(* CODESYS project MateusBastos_TalitaFelix_Versao_Final.project

Project tree, tasks and I/O mapping:
  Device : CODESYS Control Win V3, 3S - Smart Software Solutions GmbH, order no. 305021, version 3.5.11.40
    application Application
      libraries: Standard, * (System)
      task MainTask (cyclic, interval t#10ms, priority 1) calls Main_PGR
      global variables GVL
      Simulacao/
        Manual/
          program Manual_Simulacao_Silo_03 [ST]
          program Manual_Simulacao_Silo_02 [ST]
          program Manual_Simulacao_Silo_01 [ST]
        Automatico/
          program Doca2_Simulacao_Automatico [ST]
          program Doca1_Simulacao_Automatico [ST]
          program Valores_Doca2_Simulacao [ST]
          program Valores_Doca1_Simulacao [ST]
      Main/
        program Emergencia [ST]
        program Main_PGR [SFC]
      Docas/
        Manual/
          program Doca1_manual [SFC]
          program Doca2_manual [SFC]
        Automatico/
          program Doca1_automatico [SFC]
          program Doca2_automatico [SFC]
      program Alarmes [ST]
  program Valores_Simulacao_Manual [ST]
*)

// Device/Application/GVL
{attribute 'qualified_only'}
VAR_GLOBAL
// Sensores Analógicos - Entradas
LT_S01 : REAL;   // Sensor de porcentagem de etanol no silo 1
LT_S02 : REAL;   // Sensor de porcentagem de gasolina no silo 2
LT_S03 : REAL;   // Sensor de porcentagem de etanol no silo 3

// Sensores Discretos - Entradas
LSH_S01 : BOOL;  // Sensor de quantidade alta de combustível no silo 1
LSL_S01 : BOOL;  // Sensor de quantidade baixa de combustível no silo 1
LSH_S02 : BOOL;  // Sensor de quantidade alta de combustível no silo 2
LSL_S02 : BOOL;  // Sensor de quantidade baixa de combustível no silo 2
LSH_S03 : BOOL;  // Sensor de quantidade alta de combustível no silo 3
LSL_S03 : BOOL;  // Sensor de quantidade baixa de combustível no silo 3

ALARME_LSH_S01 : BOOL;  // Alarme de quantidade alta de combustível no silo 1
ALARME_LSL_S01 : BOOL;  // Alarme de quantidade baixa de combustível no silo 1
ALARME_LSH_S02 : BOOL;  // Alarme de quantidade alta de combustível no silo 2
ALARME_LSL_S02 : BOOL;  // Alarme de quantidade baixa de combustível no silo 2
ALARME_LSH_S03 : BOOL;  // Alarme de quantidade alta de combustível no silo 3
ALARME_LSL_S03 : BOOL;  // Alarme de quantidade baixa de combustível no silo 3

// Atuadores Discretos - Saídas
VA_S01 : BOOL;   // Válvula de admissão de etanol no silo 1
VA_S02 : BOOL;   // Válvula de admissão de gasolina no silo 2
VA_S03 : BOOL;   // Válvula de admissão de etanol no silo 3
VS_S01 : BOOL;   // Válvula de admissão de etanol no tanque
VS_S02_1 : BOOL; // Válvula de admissão de gasolina no tanque (primeira seção)
VS_S02_2 : BOOL; // Válvula de admissão de gasolina no tanque (segunda seção)
VS_S03 : BOOL;   // Válvula de admissão de etanol no tanque
VC_TQ2 : BOOL;   // Válvula de saída do combustível para a mangueira (tanque 2)
VC_TQ1 : BOOL;   // Válvula de saída do combustível para a mangueira (tanque 1)
M1 : BOOL;       // Misturador 1
M2 : BOOL;       // Misturador 2
B_R1 : BOOL;     // Bomba de Etanol
D1_B_R1 :BOOL;
D2_B_R1 :BOOL;
B_R2 : BOOL;
D1_B_R2 : BOOL;
D2_B_R2 : BOOL;     // Bomba de Gasolina
C_D1 : BOOL;     // Cancela 1
C_D2 : BOOL;     // Cancela 2

// Interface - máquina
liga: BOOL;
desliga: BOOL;
emergencia: BOOL;
rearme: BOOL;
Y_C_D1: BOOL;
Y_M_D1: BOOL;
Y_C_D2: BOOL;
Y_M_D2: BOOL;
etanol_D1: BOOL;
gasolina_p_D1: BOOL;
gasolina_n_D1: BOOL;
etanol_D2: BOOL;
gasolina_p_D2: BOOL;
gasolina_n_D2: BOOL;
//etanol_cheio: BOOL;
//gasolina_cheio: BOOL;
//timer_misturador: BOOL;
caminhao1_cheio: BOOL;
caminhao2_cheio: BOOL;
alarme_D1: BOOL;
alarme_D2: BOOL;

V_R_Etanol : INT := 100; //Vazao Reservatorio Etanol
V_R_Gasolina : INT := 100; //Vazao Reservatorio Gasolina
V_S01_TQ1 : INT := 50; // Vazão do Silo para o Tanque
V_S02_TQ : INT := 50; // Vazão DO Silo para o Tanque
V_S03_TQ2 : INT := 50; // Vazão DO Silo para o Tanque
TQ1_C : INT := 50;
TQ2_C : INT := 50;

volume_S01 : REAL := 50000;
volume_S02 : REAL := 50000;
volume_S03 : REAL := 50000;

volume_C1 : REAL := 0;
volume_C2 : REAL := 0;

volume_TQ1 : REAL := 0;
volume_TQ2 : REAL := 0;

volume_gasolina_C1 : REAL := 0;
volume_gasolina_C2 : REAL := 0;

volume_etanol_C1 : REAL := 0;
volume_etanol_C2 : REAL := 0;

PREMIUM : BOOL; 
ETANOL : BOOL; 

modo_op : BOOL; //Modo de operação atual do programa
switch : BOOl; //Modo de operação que o operador definiu

Transbordo_S03 : BOOL;
Transbordo_S02 : BOOL;
Transbordo_S01 : BOOL;

END_VAR

// Device/Application/Main/Main_PGR
PROGRAM Main_PGR
VAR
END_VAR

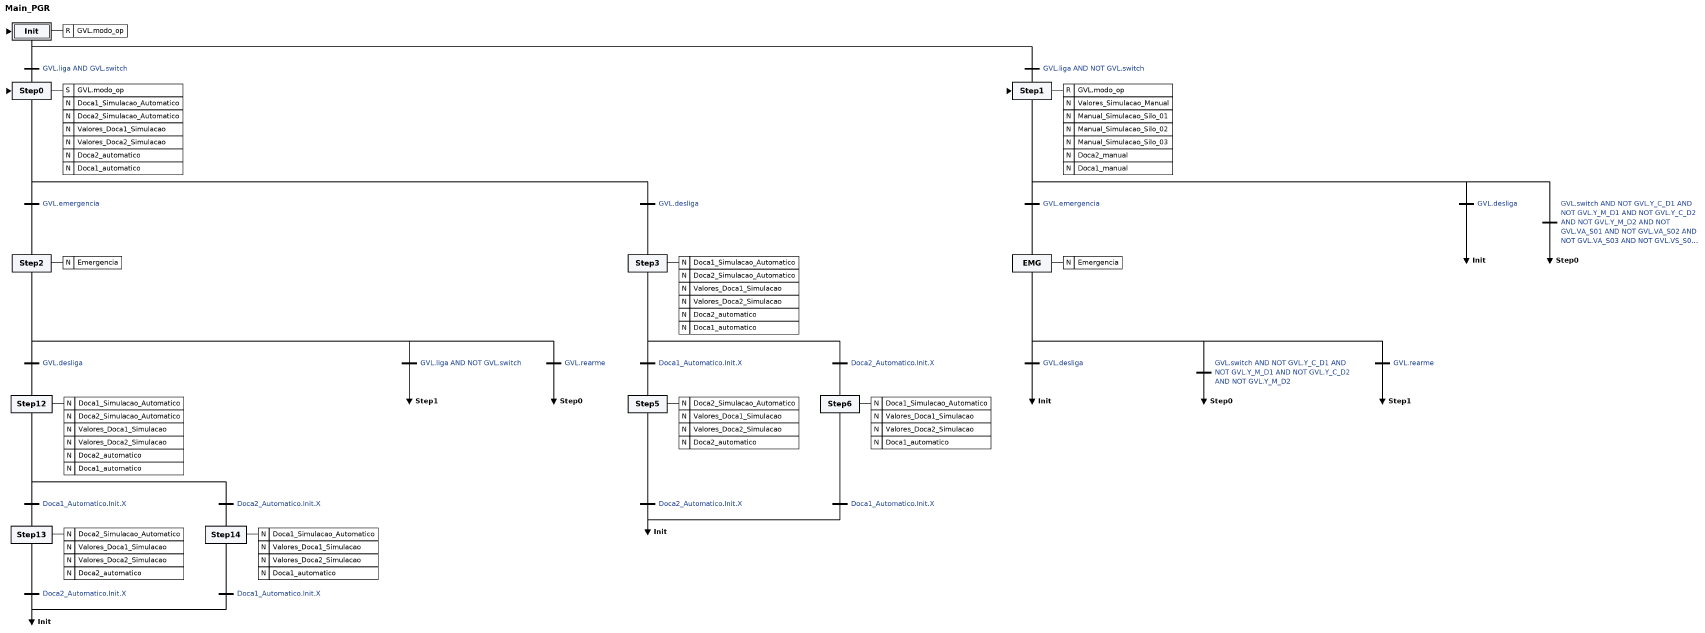
INITIAL_STEP Init:
    GVL.modo_op(R);
END_STEP
TRANSITION FROM Init TO Step0
    := GVL.liga AND GVL.switch;
END_TRANSITION
STEP Step0:
    GVL.modo_op(S);
    Doca1_Simulacao_Automatico(N);
    Doca2_Simulacao_Automatico(N);
    Valores_Doca1_Simulacao(N);
    Valores_Doca2_Simulacao(N);
    Doca2_automatico(N);
    Doca1_automatico(N);
END_STEP
TRANSITION FROM Step0 TO Step2
    := GVL.emergencia;
END_TRANSITION
STEP Step2:
    Emergencia(N);
END_STEP
TRANSITION FROM Step2 TO Step12
    := GVL.desliga;
END_TRANSITION
TRANSITION FROM Step2 TO Step1
    := GVL.liga AND NOT GVL.switch;
END_TRANSITION
TRANSITION FROM Step2 TO Step0
    := GVL.rearme;
END_TRANSITION
TRANSITION FROM Step0 TO Step3
    := GVL.desliga;
END_TRANSITION
STEP Step3:
    Doca1_Simulacao_Automatico(N);
    Doca2_Simulacao_Automatico(N);
    Valores_Doca1_Simulacao(N);
    Valores_Doca2_Simulacao(N);
    Doca2_automatico(N);
    Doca1_automatico(N);
END_STEP
TRANSITION FROM Step3 TO Step5
    := Doca1_Automatico.Init.X;
END_TRANSITION
STEP Step5:
    Doca2_Simulacao_Automatico(N);
    Valores_Doca1_Simulacao(N);
    Valores_Doca2_Simulacao(N);
    Doca2_automatico(N);
END_STEP
TRANSITION FROM Step5 TO Init
    := Doca2_Automatico.Init.X;
END_TRANSITION
TRANSITION FROM Step3 TO Step6
    := Doca2_Automatico.Init.X;
END_TRANSITION
STEP Step6:
    Doca1_Simulacao_Automatico(N);
    Valores_Doca1_Simulacao(N);
    Valores_Doca2_Simulacao(N);
    Doca1_automatico(N);
END_STEP
TRANSITION FROM Step6 TO Init
    := Doca1_Automatico.Init.X;
END_TRANSITION
TRANSITION FROM Init TO Step1
    := GVL.liga AND NOT GVL.switch;
END_TRANSITION
STEP Step1:
    GVL.modo_op(R);
    Valores_Simulacao_Manual(N);
    Manual_Simulacao_Silo_01(N);
    Manual_Simulacao_Silo_02(N);
    Manual_Simulacao_Silo_03(N);
    Doca2_manual(N);
    Doca1_manual(N);
END_STEP
TRANSITION FROM Step1 TO EMG
    := GVL.emergencia;
END_TRANSITION
STEP EMG:
    Emergencia(N);
END_STEP
TRANSITION FROM Step1 TO Init
    := GVL.desliga;
END_TRANSITION
TRANSITION FROM Step1 TO Step0
    := GVL.switch AND NOT GVL.Y_C_D1 AND NOT GVL.Y_M_D1 AND NOT GVL.Y_C_D2 AND NOT GVL.Y_M_D2 AND NOT GVL.VA_S01 AND NOT GVL.VA_S02 AND NOT GVL.VA_S03 AND NOT GVL.VS_S01 AND NOT GVL.VS_S02_1 AND NOT GVL.VS_S02_2 AND NOT GVL.VS_S03 AND NOT GVL.VC_TQ2 AND NOT GVL.VC_TQ1 AND NOT GVL.B_R2 AND NOT GVL.B_R1 AND NOT GVL.M1 AND NOT GVL.M2;
END_TRANSITION
TRANSITION FROM EMG TO Init
    := GVL.desliga;
END_TRANSITION
TRANSITION FROM EMG TO Step0
    := GVL.switch AND NOT GVL.Y_C_D1 AND NOT GVL.Y_M_D1 AND NOT GVL.Y_C_D2 AND NOT GVL.Y_M_D2;
END_TRANSITION
TRANSITION FROM EMG TO Step1
    := GVL.rearme;
END_TRANSITION
STEP Step12:
    Doca1_Simulacao_Automatico(N);
    Doca2_Simulacao_Automatico(N);
    Valores_Doca1_Simulacao(N);
    Valores_Doca2_Simulacao(N);
    Doca2_automatico(N);
    Doca1_automatico(N);
END_STEP
TRANSITION FROM Step12 TO Step13
    := Doca1_Automatico.Init.X;
END_TRANSITION
STEP Step13:
    Doca2_Simulacao_Automatico(N);
    Valores_Doca1_Simulacao(N);
    Valores_Doca2_Simulacao(N);
    Doca2_automatico(N);
END_STEP
TRANSITION FROM Step13 TO Init
    := Doca2_Automatico.Init.X;
END_TRANSITION
TRANSITION FROM Step12 TO Step14
    := Doca2_Automatico.Init.X;
END_TRANSITION
STEP Step14:
    Doca1_Simulacao_Automatico(N);
    Valores_Doca1_Simulacao(N);
    Valores_Doca2_Simulacao(N);
    Doca1_automatico(N);
END_STEP
TRANSITION FROM Step14 TO Init
    := Doca1_Automatico.Init.X;
END_TRANSITION

END_PROGRAM

// Device/Application/Simulacao/Automatico/Doca2_Simulacao_Automatico
PROGRAM Doca2_Simulacao_Automatico
VAR
END_VAR

IF NOT GVL.emergencia AND GVL.switch THEN
	//Estado  20 & //Estado 31 & //Estado 41 & //Estado 34 & //Estado 44
	IF GVL.VA_S03 AND GVL.D2_B_R1 AND NOT GVL.LSH_S03 THEN
	// Enchendo o Silo 01 de Etanol - STEP_21
		GVL.volume_S03 := GVL.volume_S03 + GVL.V_R_Etanol;
	
		GVL.volume_TQ2 := GVL.volume_TQ2;
		
		GVL.volume_C2 := GVL.volume_C2;
		
	//Estado  20	
	ELSIF GVL.VA_S02 AND (GVL.D1_B_R2 OR GVL.D2_B_R2) AND (GVL.ETANOL OR NOT GVL.Y_C_D1) AND NOT GVL.LSH_S02 THEN // Caso em que o somente a doca 2 está utilizando gasolina
		GVL.volume_S02 := GVL.volume_S02 + GVL.V_R_Gasolina;
		
	ELSIF GVL.VS_S03 AND GVL.C_D2 AND NOT GVL.VS_S02_2 AND GVL.VC_TQ2 AND GVL.volume_S03 > 0 THEN
	// Enchendo o Tanque 1 & Esvaziando o Silo 01 - STEP_20
		GVL.volume_S03 := GVL.volume_S03 - GVL.V_S03_TQ2;
		
		GVL.volume_TQ2 := GVL.volume_TQ2 + GVL.TQ2_C - GVL.V_S03_TQ2;
		
		GVL.volume_C2 := GVL.volume_C2 + GVL.TQ2_C;
		
	//Estado 30	- STEP_30 e STEP_40
	ELSIF GVL.VS_S03 AND GVL.VS_S02_2 AND GVL.C_D2 AND GVL.volume_S03 > 0 AND GVL.volume_S02 > 0 THEN
	// Enchendo o TQ 1 && Esvaziando o Silo 01 && Esvaziando o Silo 02
	
	//Situação em que começo a encher o tanque de gasolina e de etanol simultaneamente
	
		GVL.volume_S03 := GVL.volume_S03 - GVL.V_S03_TQ2; // Diminuo o volume do Silo 3
		
		GVL.volume_S02 := GVL.volume_S02 - GVL.V_S02_TQ; // Diminuo o volume do Silo 2
		
		GVL.volume_C2 := GVL.volume_C2; // Mantenho o volume do caminhão constante
		
		GVL.volume_TQ2 := GVL.volume_TQ2 + GVL.V_S02_TQ + GVL.V_S03_TQ2; // Aumento o volume do tanque 1
		
		GVL.volume_gasolina_C2 := GVL.volume_gasolina_C2 + GVL.V_S02_TQ; // Aumento a contagem da gasolina que está entrando no tanque
		
		GVL.volume_etanol_C2 := GVL.volume_etanol_C2 + GVL.V_S03_TQ2; // Aumento a contagem de etanol que está entrando no tanque
		
	//Estado 33 & Estado 43 - STEP_33
	ELSIF GVL.VS_S02_2 AND NOT GVL.VC_TQ2 AND GVL.C_D2 AND GVL.volume_S02 > 0 THEN
		GVL.volume_S02 := GVL.volume_S02 - GVL.V_S02_TQ;	
		
		GVL.volume_C2 := GVL.volume_C2;
		
		GVL.volume_TQ2 := GVL.volume_TQ2 + GVL.V_S02_TQ;
		
		GVL.volume_gasolina_C2 := GVL.volume_gasolina_C2 + GVL.V_S02_TQ;
		
	//Estado 35 & //Estado 45
	ELSIF GVL.M2 AND GVL.C_D2 THEN
		GVL.volume_C2 := GVL.volume_C2;
		GVL.volume_TQ2 := GVL.volume_TQ2;
		
	//Estado 36 & //Estado 46
	ELSIF GVL.VC_TQ2 AND GVL.C_D2 AND GVL.volume_TQ2 > 0 THEN
		GVL.volume_C2 := GVL.volume_C2 + GVL.TQ2_C;
		GVL.volume_TQ2 := GVL.volume_TQ2 - GVL.TQ2_C;
	
	ELSIF NOT GVL.Y_C_D2 AND NOT GVL.C_D2 THEN 
		GVL.volume_C2 := 0;
		GVL.volume_TQ2 := 0;
		
		Doca2_automatico.gasolina_cheio := FALSE;
		Doca2_automatico.etanol_cheio := FALSE;
		GVL.caminhao2_cheio := FALSE;
	
	END_IF
END_IF

END_PROGRAM

// Device/Application/Main/Emergencia
PROGRAM Emergencia


	GVL.VA_S01 := FALSE;   
	GVL.VA_S02 := FALSE;
	GVL.VA_S03 := FALSE;
	GVL.VS_S01 := FALSE;
	GVL.VS_S02_1 := FALSE;
	GVL.VS_S02_2 := FALSE;
	GVL.VS_S03 := FALSE;
	GVL.VC_TQ2 := FALSE;
	GVL.VC_TQ1 := FALSE;
	GVL.M1 := FALSE;
	GVL.M2 := FALSE;

END_PROGRAM

// Device/Application/Docas/Automatico/Doca2_automatico
PROGRAM Doca2_automatico
VAR_INPUT
	etanol_cheio: BOOL;
	gasolina_cheio: BOOL;
END_VAR

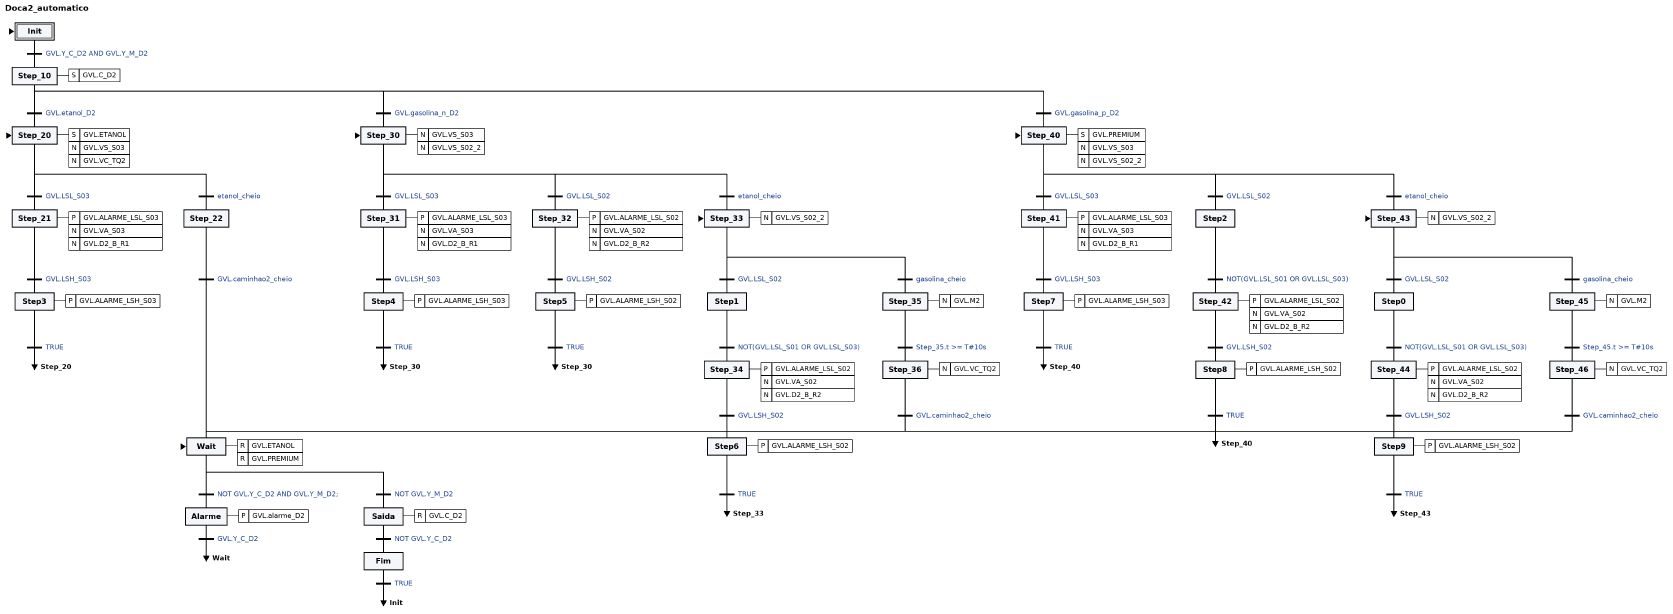
INITIAL_STEP Init:
END_STEP
TRANSITION FROM Init TO Step_10
    := GVL.Y_C_D2 AND GVL.Y_M_D2;
END_TRANSITION
STEP Step_10:
    GVL.C_D2(S);
END_STEP
TRANSITION FROM Step_10 TO Step_20
    := GVL.etanol_D2;
END_TRANSITION
STEP Step_20:
    GVL.ETANOL(S);
    GVL.VS_S03(N);
    GVL.VC_TQ2(N);
END_STEP
TRANSITION FROM Step_20 TO Step_21
    := GVL.LSL_S03;
END_TRANSITION
STEP Step_21:
    GVL.ALARME_LSL_S03(P);
    GVL.VA_S03(N);
    GVL.D2_B_R1(N);
END_STEP
TRANSITION FROM Step_21 TO Step3
    := GVL.LSH_S03;
END_TRANSITION
STEP Step3:
    GVL.ALARME_LSH_S03(P);
END_STEP
TRANSITION FROM Step3 TO Step_20
    := TRUE;
END_TRANSITION
TRANSITION FROM Step_20 TO Step_22
    := etanol_cheio;
END_TRANSITION
STEP Step_22:
END_STEP
TRANSITION FROM Step_22 TO Wait
    := GVL.caminhao2_cheio;
END_TRANSITION
TRANSITION FROM Step_10 TO Step_30
    := GVL.gasolina_n_D2;
END_TRANSITION
STEP Step_30:
    GVL.VS_S03(N);
    GVL.VS_S02_2(N);
END_STEP
TRANSITION FROM Step_30 TO Step_31
    := GVL.LSL_S03;
END_TRANSITION
STEP Step_31:
    GVL.ALARME_LSL_S03(P);
    GVL.VA_S03(N);
    GVL.D2_B_R1(N);
END_STEP
TRANSITION FROM Step_31 TO Step4
    := GVL.LSH_S03;
END_TRANSITION
STEP Step4:
    GVL.ALARME_LSH_S03(P);
END_STEP
TRANSITION FROM Step4 TO Step_30
    := TRUE;
END_TRANSITION
TRANSITION FROM Step_30 TO Step_32
    := GVL.LSL_S02;
END_TRANSITION
STEP Step_32:
    GVL.ALARME_LSL_S02(P);
    GVL.VA_S02(N);
    GVL.D2_B_R2(N);
END_STEP
TRANSITION FROM Step_32 TO Step5
    := GVL.LSH_S02;
END_TRANSITION
STEP Step5:
    GVL.ALARME_LSH_S02(P);
END_STEP
TRANSITION FROM Step5 TO Step_30
    := TRUE;
END_TRANSITION
TRANSITION FROM Step_30 TO Step_33
    := etanol_cheio;
END_TRANSITION
STEP Step_33:
    GVL.VS_S02_2(N);
END_STEP
TRANSITION FROM Step_33 TO Step1
    := GVL.LSL_S02;
END_TRANSITION
STEP Step1:
END_STEP
TRANSITION FROM Step1 TO Step_34
    := NOT(GVL.LSL_S01 OR GVL.LSL_S03);
END_TRANSITION
STEP Step_34:
    GVL.ALARME_LSL_S02(P);
    GVL.VA_S02(N);
    GVL.D2_B_R2(N);
END_STEP
TRANSITION FROM Step_34 TO Step6
    := GVL.LSH_S02;
END_TRANSITION
STEP Step6:
    GVL.ALARME_LSH_S02(P);
END_STEP
TRANSITION FROM Step6 TO Step_33
    := TRUE;
END_TRANSITION
TRANSITION FROM Step_33 TO Step_35
    := gasolina_cheio;
END_TRANSITION
STEP Step_35:
    GVL.M2(N);
END_STEP
TRANSITION FROM Step_35 TO Step_36
    := Step_35.t >= T#10s;
END_TRANSITION
STEP Step_36:
    GVL.VC_TQ2(N);
END_STEP
TRANSITION FROM Step_36 TO Wait
    := GVL.caminhao2_cheio;
END_TRANSITION
TRANSITION FROM Step_10 TO Step_40
    := GVL.gasolina_p_D2;
END_TRANSITION
STEP Step_40:
    GVL.PREMIUM(S);
    GVL.VS_S03(N);
    GVL.VS_S02_2(N);
END_STEP
TRANSITION FROM Step_40 TO Step_41
    := GVL.LSL_S03;
END_TRANSITION
STEP Step_41:
    GVL.ALARME_LSL_S03(P);
    GVL.VA_S03(N);
    GVL.D2_B_R1(N);
END_STEP
TRANSITION FROM Step_41 TO Step7
    := GVL.LSH_S03;
END_TRANSITION
STEP Step7:
    GVL.ALARME_LSH_S03(P);
END_STEP
TRANSITION FROM Step7 TO Step_40
    := TRUE;
END_TRANSITION
TRANSITION FROM Step_40 TO Step2
    := GVL.LSL_S02;
END_TRANSITION
STEP Step2:
END_STEP
TRANSITION FROM Step2 TO Step_42
    := NOT(GVL.LSL_S01 OR GVL.LSL_S03);
END_TRANSITION
STEP Step_42:
    GVL.ALARME_LSL_S02(P);
    GVL.VA_S02(N);
    GVL.D2_B_R2(N);
END_STEP
TRANSITION FROM Step_42 TO Step8
    := GVL.LSH_S02;
END_TRANSITION
STEP Step8:
    GVL.ALARME_LSH_S02(P);
END_STEP
TRANSITION FROM Step8 TO Step_40
    := TRUE;
END_TRANSITION
TRANSITION FROM Step_40 TO Step_43
    := etanol_cheio;
END_TRANSITION
STEP Step_43:
    GVL.VS_S02_2(N);
END_STEP
TRANSITION FROM Step_43 TO Step0
    := GVL.LSL_S02;
END_TRANSITION
STEP Step0:
END_STEP
TRANSITION FROM Step0 TO Step_44
    := NOT(GVL.LSL_S01 OR GVL.LSL_S03);
END_TRANSITION
STEP Step_44:
    GVL.ALARME_LSL_S02(P);
    GVL.VA_S02(N);
    GVL.D2_B_R2(N);
END_STEP
TRANSITION FROM Step_44 TO Step9
    := GVL.LSH_S02;
END_TRANSITION
STEP Step9:
    GVL.ALARME_LSH_S02(P);
END_STEP
TRANSITION FROM Step9 TO Step_43
    := TRUE;
END_TRANSITION
TRANSITION FROM Step_43 TO Step_45
    := gasolina_cheio;
END_TRANSITION
STEP Step_45:
    GVL.M2(N);
END_STEP
TRANSITION FROM Step_45 TO Step_46
    := Step_45.t >= T#10s;
END_TRANSITION
STEP Step_46:
    GVL.VC_TQ2(N);
END_STEP
TRANSITION FROM Step_46 TO Wait
    := GVL.caminhao2_cheio;
END_TRANSITION
STEP Wait:
    GVL.ETANOL(R);
    GVL.PREMIUM(R);
END_STEP
TRANSITION FROM Wait TO Alarme
    := NOT GVL.Y_C_D2 AND GVL.Y_M_D2;
END_TRANSITION
STEP Alarme:
    GVL.alarme_D2(P);
END_STEP
TRANSITION FROM Alarme TO Wait
    := GVL.Y_C_D2;
END_TRANSITION
TRANSITION FROM Wait TO Saida
    := NOT GVL.Y_M_D2;
END_TRANSITION
STEP Saida:
    GVL.C_D2(R);
END_STEP
TRANSITION FROM Saida TO Fim
    := NOT GVL.Y_C_D2;
END_TRANSITION
STEP Fim:
END_STEP
TRANSITION FROM Fim TO Init
    := TRUE;
END_TRANSITION

END_PROGRAM

// Device/Application/Docas/Manual/Doca1_manual
PROGRAM Doca1_manual
VAR_INPUT
	Ligar : BOOL;
END_VAR

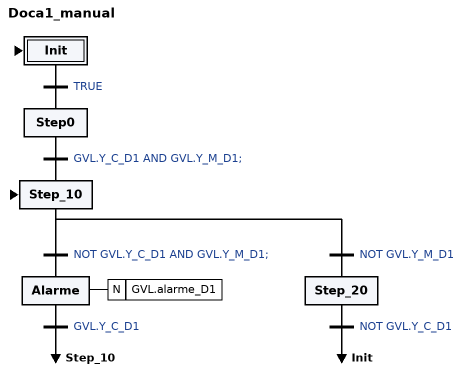
INITIAL_STEP Init:
END_STEP
TRANSITION FROM Init TO Step0
    := TRUE;
END_TRANSITION
STEP Step0:
END_STEP
TRANSITION FROM Step0 TO Step_10
    := GVL.Y_C_D1 AND GVL.Y_M_D1;
END_TRANSITION
STEP Step_10:
END_STEP
TRANSITION FROM Step_10 TO Alarme
    := NOT GVL.Y_C_D1 AND GVL.Y_M_D1;
END_TRANSITION
STEP Alarme:
    GVL.alarme_D1(N);
END_STEP
TRANSITION FROM Alarme TO Step_10
    := GVL.Y_C_D1;
END_TRANSITION
TRANSITION FROM Step_10 TO Step_20
    := NOT GVL.Y_M_D1;
END_TRANSITION
STEP Step_20:
END_STEP
TRANSITION FROM Step_20 TO Init
    := NOT GVL.Y_C_D1;
END_TRANSITION

END_PROGRAM

// Device/Application/Docas/Manual/Doca2_manual
PROGRAM Doca2_manual

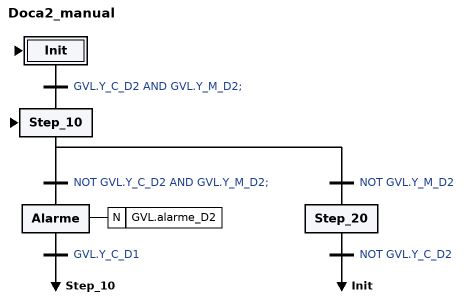
INITIAL_STEP Init:
END_STEP
TRANSITION FROM Init TO Step_10
    := GVL.Y_C_D2 AND GVL.Y_M_D2;
END_TRANSITION
STEP Step_10:
END_STEP
TRANSITION FROM Step_10 TO Alarme
    := NOT GVL.Y_C_D2 AND GVL.Y_M_D2;
END_TRANSITION
STEP Alarme:
    GVL.alarme_D2(N);
END_STEP
TRANSITION FROM Alarme TO Step_10
    := GVL.Y_C_D1;
END_TRANSITION
TRANSITION FROM Step_10 TO Step_20
    := NOT GVL.Y_M_D2;
END_TRANSITION
STEP Step_20:
END_STEP
TRANSITION FROM Step_20 TO Init
    := NOT GVL.Y_C_D2;
END_TRANSITION

END_PROGRAM

// Device/Application/Docas/Automatico/Doca1_automatico
PROGRAM Doca1_automatico

VAR_INPUT
	etanol_cheio: BOOL;
	gasolina_cheio: BOOL;
END_VAR

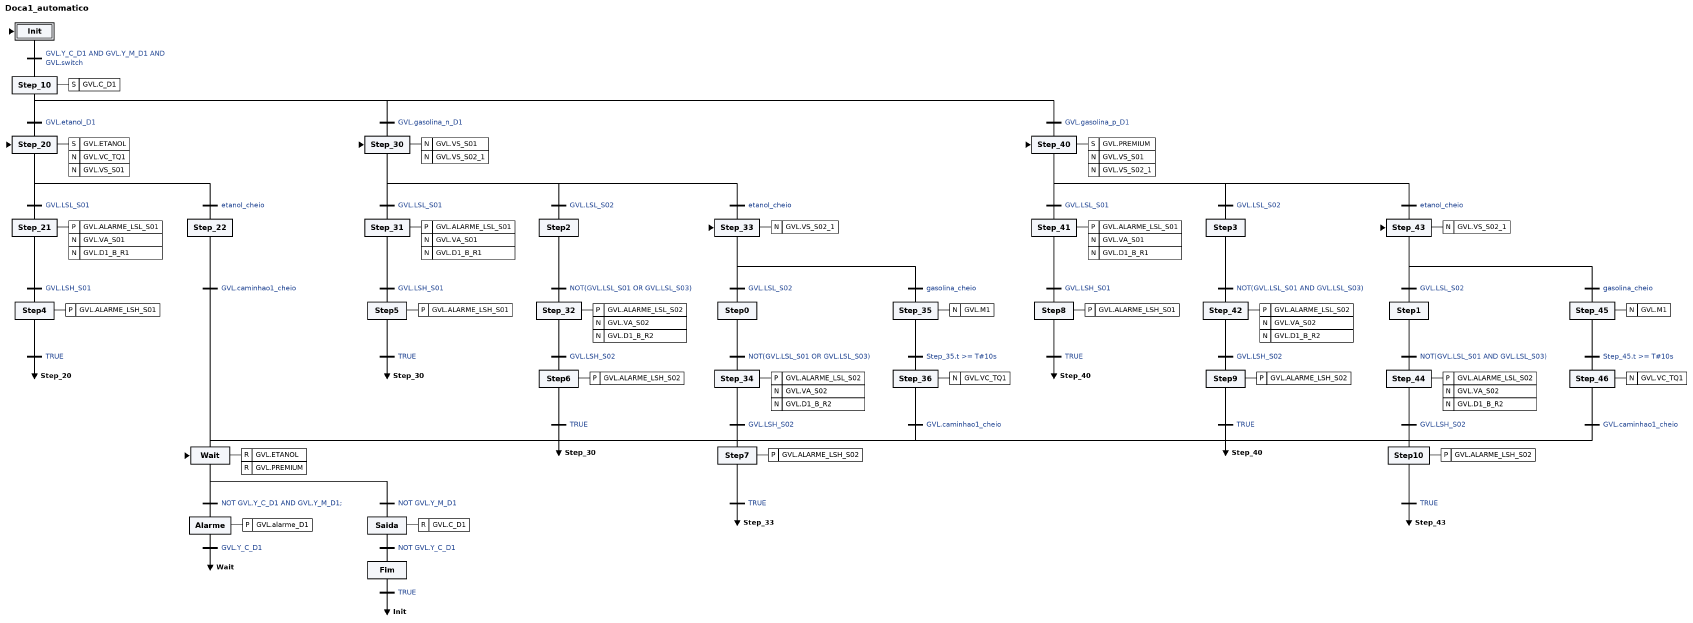
INITIAL_STEP Init:
END_STEP
TRANSITION FROM Init TO Step_10
    := GVL.Y_C_D1 AND GVL.Y_M_D1 AND GVL.switch;
END_TRANSITION
STEP Step_10:
    GVL.C_D1(S);
END_STEP
TRANSITION FROM Step_10 TO Step_20
    := GVL.etanol_D1;
END_TRANSITION
STEP Step_20:
    GVL.ETANOL(S);
    GVL.VC_TQ1(N);
    GVL.VS_S01(N);
END_STEP
TRANSITION FROM Step_20 TO Step_21
    := GVL.LSL_S01;
END_TRANSITION
STEP Step_21:
    GVL.ALARME_LSL_S01(P);
    GVL.VA_S01(N);
    GVL.D1_B_R1(N);
END_STEP
TRANSITION FROM Step_21 TO Step4
    := GVL.LSH_S01;
END_TRANSITION
STEP Step4:
    GVL.ALARME_LSH_S01(P);
END_STEP
TRANSITION FROM Step4 TO Step_20
    := TRUE;
END_TRANSITION
TRANSITION FROM Step_20 TO Step_22
    := etanol_cheio;
END_TRANSITION
STEP Step_22:
END_STEP
TRANSITION FROM Step_22 TO Wait
    := GVL.caminhao1_cheio;
END_TRANSITION
TRANSITION FROM Step_10 TO Step_30
    := GVL.gasolina_n_D1;
END_TRANSITION
STEP Step_30:
    GVL.VS_S01(N);
    GVL.VS_S02_1(N);
END_STEP
TRANSITION FROM Step_30 TO Step_31
    := GVL.LSL_S01;
END_TRANSITION
STEP Step_31:
    GVL.ALARME_LSL_S01(P);
    GVL.VA_S01(N);
    GVL.D1_B_R1(N);
END_STEP
TRANSITION FROM Step_31 TO Step5
    := GVL.LSH_S01;
END_TRANSITION
STEP Step5:
    GVL.ALARME_LSH_S01(P);
END_STEP
TRANSITION FROM Step5 TO Step_30
    := TRUE;
END_TRANSITION
TRANSITION FROM Step_30 TO Step2
    := GVL.LSL_S02;
END_TRANSITION
STEP Step2:
END_STEP
TRANSITION FROM Step2 TO Step_32
    := NOT(GVL.LSL_S01 OR GVL.LSL_S03);
END_TRANSITION
STEP Step_32:
    GVL.ALARME_LSL_S02(P);
    GVL.VA_S02(N);
    GVL.D1_B_R2(N);
END_STEP
TRANSITION FROM Step_32 TO Step6
    := GVL.LSH_S02;
END_TRANSITION
STEP Step6:
    GVL.ALARME_LSH_S02(P);
END_STEP
TRANSITION FROM Step6 TO Step_30
    := TRUE;
END_TRANSITION
TRANSITION FROM Step_30 TO Step_33
    := etanol_cheio;
END_TRANSITION
STEP Step_33:
    GVL.VS_S02_1(N);
END_STEP
TRANSITION FROM Step_33 TO Step0
    := GVL.LSL_S02;
END_TRANSITION
STEP Step0:
END_STEP
TRANSITION FROM Step0 TO Step_34
    := NOT(GVL.LSL_S01 OR GVL.LSL_S03);
END_TRANSITION
STEP Step_34:
    GVL.ALARME_LSL_S02(P);
    GVL.VA_S02(N);
    GVL.D1_B_R2(N);
END_STEP
TRANSITION FROM Step_34 TO Step7
    := GVL.LSH_S02;
END_TRANSITION
STEP Step7:
    GVL.ALARME_LSH_S02(P);
END_STEP
TRANSITION FROM Step7 TO Step_33
    := TRUE;
END_TRANSITION
TRANSITION FROM Step_33 TO Step_35
    := gasolina_cheio;
END_TRANSITION
STEP Step_35:
    GVL.M1(N);
END_STEP
TRANSITION FROM Step_35 TO Step_36
    := Step_35.t >= T#10s;
END_TRANSITION
STEP Step_36:
    GVL.VC_TQ1(N);
END_STEP
TRANSITION FROM Step_36 TO Wait
    := GVL.caminhao1_cheio;
END_TRANSITION
TRANSITION FROM Step_10 TO Step_40
    := GVL.gasolina_p_D1;
END_TRANSITION
STEP Step_40:
    GVL.PREMIUM(S);
    GVL.VS_S01(N);
    GVL.VS_S02_1(N);
END_STEP
TRANSITION FROM Step_40 TO Step_41
    := GVL.LSL_S01;
END_TRANSITION
STEP Step_41:
    GVL.ALARME_LSL_S01(P);
    GVL.VA_S01(N);
    GVL.D1_B_R1(N);
END_STEP
TRANSITION FROM Step_41 TO Step8
    := GVL.LSH_S01;
END_TRANSITION
STEP Step8:
    GVL.ALARME_LSH_S01(P);
END_STEP
TRANSITION FROM Step8 TO Step_40
    := TRUE;
END_TRANSITION
TRANSITION FROM Step_40 TO Step3
    := GVL.LSL_S02;
END_TRANSITION
STEP Step3:
END_STEP
TRANSITION FROM Step3 TO Step_42
    := NOT(GVL.LSL_S01 AND GVL.LSL_S03);
END_TRANSITION
STEP Step_42:
    GVL.ALARME_LSL_S02(P);
    GVL.VA_S02(N);
    GVL.D1_B_R2(N);
END_STEP
TRANSITION FROM Step_42 TO Step9
    := GVL.LSH_S02;
END_TRANSITION
STEP Step9:
    GVL.ALARME_LSH_S02(P);
END_STEP
TRANSITION FROM Step9 TO Step_40
    := TRUE;
END_TRANSITION
TRANSITION FROM Step_40 TO Step_43
    := etanol_cheio;
END_TRANSITION
STEP Step_43:
    GVL.VS_S02_1(N);
END_STEP
TRANSITION FROM Step_43 TO Step1
    := GVL.LSL_S02;
END_TRANSITION
STEP Step1:
END_STEP
TRANSITION FROM Step1 TO Step_44
    := NOT(GVL.LSL_S01 AND GVL.LSL_S03);
END_TRANSITION
STEP Step_44:
    GVL.ALARME_LSL_S02(P);
    GVL.VA_S02(N);
    GVL.D1_B_R2(N);
END_STEP
TRANSITION FROM Step_44 TO Step10
    := GVL.LSH_S02;
END_TRANSITION
STEP Step10:
    GVL.ALARME_LSH_S02(P);
END_STEP
TRANSITION FROM Step10 TO Step_43
    := TRUE;
END_TRANSITION
TRANSITION FROM Step_43 TO Step_45
    := gasolina_cheio;
END_TRANSITION
STEP Step_45:
    GVL.M1(N);
END_STEP
TRANSITION FROM Step_45 TO Step_46
    := Step_45.t >= T#10s;
END_TRANSITION
STEP Step_46:
    GVL.VC_TQ1(N);
END_STEP
TRANSITION FROM Step_46 TO Wait
    := GVL.caminhao1_cheio;
END_TRANSITION
STEP Wait:
    GVL.ETANOL(R);
    GVL.PREMIUM(R);
END_STEP
TRANSITION FROM Wait TO Alarme
    := NOT GVL.Y_C_D1 AND GVL.Y_M_D1;
END_TRANSITION
STEP Alarme:
    GVL.alarme_D1(P);
END_STEP
TRANSITION FROM Alarme TO Wait
    := GVL.Y_C_D1;
END_TRANSITION
TRANSITION FROM Wait TO Saida
    := NOT GVL.Y_M_D1;
END_TRANSITION
STEP Saida:
    GVL.C_D1(R);
END_STEP
TRANSITION FROM Saida TO Fim
    := NOT GVL.Y_C_D1;
END_TRANSITION
STEP Fim:
END_STEP
TRANSITION FROM Fim TO Init
    := TRUE;
END_TRANSITION

END_PROGRAM

// Device/Application/Simulacao/Manual/Manual_Simulacao_Silo_03
PROGRAM Manual_Simulacao_Silo_03
VAR
END_VAR

IF NOT GVL.emergencia AND NOT GVL.switch THEN
	
	IF NOT GVL.D1_B_R1 AND NOT GVL.VS_S03 AND GVL.VC_TQ2 THEN
	
		IF GVL.volume_TQ2 > 0 THEN
			
			GVL.volume_TQ2 := GVL.volume_TQ2 - GVL.TQ2_C; // Diminuo o volume do tanque
			
		END_IF
		
	ELSIF NOT GVL.D2_B_R1 AND GVL.VS_S03 AND NOT GVL.VC_TQ2 THEN
		
		IF GVL.volume_S03 > 0 AND GVL.volume_TQ2 <= 50000 THEN
			GVL.volume_S03 := GVL.volume_S03 - GVL.V_S03_TQ2; //Diminuo o volume do silo
		
			GVL.volume_TQ2 := GVL.volume_TQ2 + GVL.V_S03_TQ2; // Aumento o volume do tanque
		END_IF
	
	ELSIF NOT GVL.D2_B_R1 AND GVL.VS_S03 AND GVL.VC_TQ2 THEN
		
		IF GVL.volume_S03 > 0 THEN
			GVL.volume_S03 := GVL.volume_S03 - GVL.V_S03_TQ2; //Diminuo o volume do silo
			GVL.volume_TQ2 := GVL.volume_TQ2 + GVL.V_S03_TQ2 - GVL.TQ2_C;;
		ELSIF GVL.volume_TQ2 > 0 THEN
			GVL.volume_TQ2 := GVL.volume_TQ2 - GVL.TQ2_C; // Mantenho o volume do tanque, 
		END_IF
		
	ELSIF GVL.D2_B_R1 AND NOT GVL.VA_S03 AND NOT GVL.VS_S03 AND GVL.VC_TQ2 THEN
		
		IF GVL.volume_TQ2 > 0 THEN
			
			GVL.volume_TQ2 := GVL.volume_TQ2 - GVL.TQ2_C; // Diminuo o volume do tanque
			
		END_IF
		
	ELSIF GVL.D2_B_R1 AND NOT GVL.VA_S03 AND GVL.VS_S03 AND NOT GVL.VC_TQ2 THEN
	
		IF GVL.volume_S03 > 0 AND GVL.volume_TQ2 <= 50000 THEN
			
			GVL.volume_S03 := GVL.volume_S03 - GVL.V_S03_TQ2; //Diminuo o volume do silo
		
			GVL.volume_TQ2 := GVL.volume_TQ2 + GVL.V_S03_TQ2; // Aumento o volume do tanque
		END_IF
	
	ELSIF GVL.D2_B_R1 AND NOT GVL.VA_S03 AND GVL.VS_S03 AND GVL.VC_TQ2 THEN
	
		IF GVL.volume_S03 > 0 THEN
			GVL.volume_S03 := GVL.volume_S03 - GVL.V_S03_TQ2; //Diminuo o volume do silo
			GVL.volume_TQ1 := GVL.volume_TQ1 + GVL.V_S03_TQ2 - GVL.TQ2_C;;
		ELSIF GVL.volume_TQ1 > 0 THEN
			GVL.volume_TQ2 := GVL.volume_TQ2 - GVL.TQ2_C; // Mantenho o volume do tanque, 
		END_IF	
		
	ELSIF GVL.D2_B_R1 AND GVL.VA_S03 AND NOT GVL.VS_S03 AND NOT GVL.VC_TQ2 THEN	
		IF GVL.volume_S03 < 50000 THEN		
			GVL.volume_S03 := GVL.volume_S03 + GVL.V_S03_TQ2;
		ELSIF GVL.volume_S03 > 50000 THEN
			GVL.Transbordo_S03 := TRUE;
		END_IF
		
	ELSIF GVL.D2_B_R1 AND GVL.VA_S03 AND NOT GVL.VS_S03 AND NOT GVL.VC_TQ2 THEN	
		IF GVL.volume_S03 < 50000 THEN		
			GVL.volume_S03 := GVL.volume_S03 + GVL.V_S03_TQ2;
		ELSIF GVL.volume_S03 > 50000 THEN
			GVL.Transbordo_S03 := TRUE;
		END_IF
		
	ELSIF GVL.D2_B_R1 AND GVL.VA_S03 AND NOT GVL.VS_S03 AND GVL.VC_TQ2 THEN	
		
		IF GVL.volume_S03 < 50000 AND GVL.volume_TQ2 > 0 THEN	
	
			GVL.volume_S03 := GVL.volume_S03 + GVL.V_R_Etanol;
			GVL.volume_TQ2 := GVL.volume_TQ2 - GVL.TQ2_C;
			
		ELSIF GVL.volume_S03 < 50000 AND GVL.volume_TQ2 < 0 THEN
			
			GVL.volume_S03 := GVL.volume_S03 + GVL.V_R_Etanol;
			
		ELSIF GVL.volume_S03 > 50000 AND GVL.volume_TQ2 > 0 THEN
			
			GVL.Transbordo_S03 := TRUE;
			GVL.volume_TQ2 := GVL.volume_TQ2 - GVL.TQ2_C;
			
		ELSIF GVL.volume_S03 > 50000  AND GVL.volume_TQ2 < 0 THEN
			GVL.Transbordo_S03 := TRUE;
		END_IF
	
	ELSIF GVL.D2_B_R1 AND GVL.VA_S03 AND GVL.VS_S03 AND NOT GVL.VC_TQ2 THEN	
		
		IF GVL.volume_S03 < 50000 AND GVL.volume_TQ2 < 25000  THEN	
	
			GVL.volume_S03 := GVL.volume_S03 + GVL.V_R_Etanol;
			GVL.volume_S03 := GVL.volume_S03 - GVL.V_S03_TQ2;
			GVL.volume_TQ2 := GVL.volume_TQ2 + GVL.V_S03_TQ2;
			
		ELSIF GVL.volume_S03 > 50000 AND GVL.volume_TQ2 < 25000  THEN	
			
			GVL.Transbordo_S03 := TRUE;
			GVL.volume_TQ2 := GVL.volume_TQ2 + GVL.V_S03_TQ2;
			
		ELSIF GVL.volume_S03 < 50000 AND GVL.volume_TQ2 > 25000 THEN
			
			GVL.volume_S03 := GVL.volume_S03 + GVL.V_R_Etanol;
			
		ELSIF GVL.volume_S03 > 50000 AND GVL.volume_TQ2 >25000 THEN
			
			GVL.Transbordo_S03 := TRUE;
			
		END_IF
	
	ELSIF GVL.D2_B_R1 AND GVL.VA_S03 AND GVL.VS_S03 AND GVL.VC_TQ2 THEN		
		
		IF GVL.volume_S03 < 50000 AND GVL.volume_TQ2 < 25000  THEN	
	
			GVL.volume_S03 := GVL.volume_S03 + GVL.V_R_Etanol;
			GVL.volume_S03 := GVL.volume_S03 - GVL.V_S03_TQ2;
			GVL.volume_TQ2 := GVL.volume_TQ2 + GVL.V_S03_TQ2;
			GVL.volume_TQ2 := GVL.volume_TQ2 - GVL.TQ2_C;
			
		ELSIF GVL.volume_S03 > 50000 AND GVL.volume_TQ2 < 25000  THEN	
			
			GVL.Transbordo_S03 := TRUE;
			GVL.volume_TQ2 := GVL.volume_TQ2 + GVL.V_S03_TQ2;
			GVL.volume_TQ2 := GVL.volume_TQ2 - GVL.TQ2_C;
			
		ELSIF GVL.volume_S03 < 50000 AND GVL.volume_TQ2 > 25000 THEN
			
			GVL.volume_S03:= GVL.volume_S03 + GVL.V_R_Etanol;
			
		ELSIF GVL.volume_S03 > 50000 AND GVL.volume_TQ2 >25000 THEN
			
			GVL.Transbordo_S03 := TRUE;
			
		END_IF
		
	END_IF
END_IF

IF GVL.volume_S03 > 45000 AND GVL.VA_S03 AND (GVL.D1_B_R1 OR GVL.D1_B_R1) THEN
	
	GVL.LSH_S03 := TRUE;
	GVL.LSL_S03 := FALSE;
	
	GVL.ALARME_LSH_S03 := TRUE;
	GVL.ALARME_LSL_S03 := FALSE;
	
ELSIF GVL.volume_S03 < 5000 THEN
	
	GVL.LSH_S03 := FALSE;
	GVL.LSL_S03 := TRUE;
	
	GVL.ALARME_LSH_S03 := FALSE;
	GVL.ALARME_LSL_S03 := TRUE;
	
END_IF

IF (GVL.D1_B_R1 OR GVL.D2_B_R1) THEN
	GVL.B_R1 := TRUE;
ELSE
	GVL.B_R1 := FALSE;
END_IF

IF (GVL.D1_B_R2 OR GVL.D2_B_R2) THEN
	GVL.B_R2 := TRUE;
ELSE
	GVL.B_R2 := FALSE;
END_IF

END_PROGRAM

// Device/Application/Simulacao/Automatico/Doca1_Simulacao_Automatico
PROGRAM Doca1_Simulacao_Automatico
VAR
END_VAR

IF NOT GVL.emergencia AND GVL.switch THEN
	//Estado  20 & //Estado 31 & //Estado 41 & //Estado 34 & //Estado 44
	IF GVL.VA_S01 AND GVL.D1_B_R1 AND NOT GVL.LSH_S01 AND NOT(GVL.volume_S01 > 50000) THEN
	// Enchendo o Silo 01 de Etanol - STEP_21
		GVL.volume_S01 := GVL.volume_S01 + GVL.V_R_Etanol;
	
		GVL.volume_TQ1 := GVL.volume_TQ1;
		
		GVL.volume_C1 := GVL.volume_C1;
		
	ELSIF GVL.VA_S02 AND (GVL.D2_B_R2 OR GVL.D1_B_R2) AND NOT GVL.LSH_S02 THEN
	// Enchendo o Silo de Gasolina
		GVL.volume_S02 := GVL.volume_S02 + GVL.V_R_Gasolina;
		
	//Estado  21	
	ELSIF GVL.VS_S01 AND GVL.C_D1 AND NOT GVL.VS_S02_1 AND GVL.VC_TQ1 AND GVL.volume_S01 > 0 THEN
	// Enchendo o Tanque 1 & Esvaziando o Silo 01 - STEP_20
		GVL.volume_S01 := GVL.volume_S01 - GVL.V_S01_TQ1;
		
		GVL.volume_TQ1 := GVL.volume_TQ1 + GVL.TQ1_C - GVL.V_S01_TQ1;
		
		GVL.volume_C1 := GVL.volume_C1 + GVL.TQ1_C;
		
	//Estado 30	- STEP_30
	ELSIF GVL.VS_S01 AND GVL.VS_S02_1 AND GVL.C_D1 AND GVL.volume_S01 > 0 AND GVL.volume_S02 > 0 THEN
	// Enchendo o TQ 1 && Esvaziando o Silo 01 && Esvaziando o Silo 02
	
	//Situação em que começo a encher o tanque de gasolina e de etanol simultaneamente
	
		GVL.volume_S01 := GVL.volume_S01 - GVL.V_S01_TQ1; // Diminuo o volume do Silo 1
		
		GVL.volume_S02 := GVL.volume_S02 - GVL.V_S02_TQ; // Diminuo o volume do Silo 2
		
		GVL.volume_C1 := GVL.volume_C1; // Mantenho o volume do caminhão constante
		
		GVL.volume_TQ1 := GVL.volume_TQ1 + GVL.V_S02_TQ + GVL.V_S01_TQ1; // Aumento o volume do tanque 1
		
		GVL.volume_gasolina_C1 := GVL.volume_gasolina_C1 + GVL.V_S02_TQ; // Aumento a contagem da gasolina que está entrando no tanque
		
		GVL.volume_etanol_C1 := GVL.volume_etanol_C1 + GVL.V_S01_TQ1; // Aumento a contagem de etanol que está entrando no tanque
		
	//Estado 33 & Estado 43 - STEP_33
	ELSIF GVL.VS_S02_1 AND NOT GVL.VC_TQ1 AND GVL.C_D1 AND GVL.volume_S02 > 0 THEN
		GVL.volume_S02 := GVL.volume_S02 - GVL.V_S02_TQ;	
		
		GVL.volume_C1 := GVL.volume_C1;
		
		GVL.volume_TQ1 := GVL.volume_TQ1 + GVL.V_S02_TQ;
		
		GVL.volume_gasolina_C1 := GVL.volume_gasolina_C1 + GVL.V_S02_TQ;
		
	//Estado 35 & //Estado 45
	ELSIF GVL.M1 AND GVL.C_D1 THEN
		GVL.volume_C1 := GVL.volume_C1;
		GVL.volume_TQ1 := GVL.volume_TQ1;
		
	//Estado 36 & //Estado 46
	ELSIF GVL.VC_TQ1 AND GVL.C_D1 AND GVL.volume_TQ1 > 0 THEN
		GVL.volume_C1 := GVL.volume_C1 + GVL.TQ1_C;
		GVL.volume_TQ1 := GVL.volume_TQ1 - GVL.TQ1_C;
	
	ELSIF NOT GVL.Y_C_D1 AND NOT GVL.C_D1 THEN 
		GVL.volume_C1 := 0;
		GVL.volume_TQ1 := 0;
		
		Doca1_automatico.gasolina_cheio := FALSE;
		Doca1_automatico.etanol_cheio := FALSE;
		GVL.caminhao1_cheio := FALSE;
		
	END_IF
END_IF

END_PROGRAM

// Device/Application/Simulacao/Manual/Manual_Simulacao_Silo_02
PROGRAM Manual_Simulacao_Silo_02
VAR
END_VAR

IF NOT GVL.emergencia THEN
	
	IF NOT (GVL.D1_B_R2 AND GVL.D2_B_R2) AND NOT GVL.VS_S02_1 AND GVL.VS_S02_2 THEN
	
		IF GVL.volume_S02 > 0 AND GVL.volume_TQ2 < 25000 THEN
			GVL.volume_S02 := GVL.volume_S02 - GVL.V_S02_TQ;
			GVL.volume_TQ2 := GVL.volume_TQ2 + GVL.V_S02_TQ; // Diminuo o volume do tanque
			
		ELSIF GVL.volume_S02 > 0 AND GVL.volume_TQ2 >= 25000 THEN
			GVL.volume_S02 := GVL.volume_S02 - GVL.V_S02_TQ;
		END_IF
		
	ELSIF NOT GVL.D1_B_R2 AND GVL.VS_S02_1 AND NOT GVL.VS_S02_2 THEN
	
		IF GVL.volume_S02 > 0 AND GVL.volume_TQ1 < 25000 THEN
			GVL.volume_S02 := GVL.volume_S02 - GVL.V_S02_TQ;
			GVL.volume_TQ1 := GVL.volume_TQ1 + GVL.V_S02_TQ; // Diminuo o volume do tanque
			
		ELSIF GVL.volume_S02 > 0 AND GVL.volume_TQ1 >= 25000 THEN
			GVL.volume_S02 := GVL.volume_S02 - GVL.V_S02_TQ;
		END_IF
	
	ELSIF NOT (GVL.D1_B_R2 AND GVL.D2_B_R2) AND GVL.VS_S02_1 AND GVL.VS_S02_2 THEN
		
			IF GVL.volume_S02 > 0 AND GVL.volume_TQ1 < 25000 AND GVL.volume_TQ2 < 25000 THEN
				GVL.volume_S02 := GVL.volume_S02 - GVL.V_S02_TQ;
				GVL.volume_TQ1 := GVL.volume_TQ1 + GVL.V_S02_TQ; // Diminuo o volume do tanque
				GVL.volume_TQ2 := GVL.volume_TQ2 + GVL.V_S02_TQ;
				
			ELSIF GVL.volume_S02 > 0 AND GVL.volume_TQ1 >= 25000 AND GVL.volume_TQ2 < 25000 THEN
				GVL.volume_S02 := GVL.volume_S02 - GVL.V_S02_TQ;
				GVL.volume_TQ2 := GVL.volume_TQ2 + GVL.V_S02_TQ;
				
			ELSIF GVL.volume_S02 > 0 AND GVL.volume_TQ1 < 25000 AND GVL.volume_TQ2 >= 25000 THEN
				GVL.volume_S02 := GVL.volume_S02 - GVL.V_S02_TQ;
				GVL.volume_TQ1 := GVL.volume_TQ1 + GVL.V_S02_TQ;
				
			ELSIF GVL.volume_S02 > 0 AND GVL.volume_TQ1 >= 25000 AND GVL.volume_TQ2 >= 25000 THEN
				GVL.volume_S02 := GVL.volume_S02 - GVL.V_S02_TQ;
				
			END_IF
	
	ELSIF (GVL.D1_B_R2 OR GVL.D2_B_R2) AND NOT GVL.VA_S02  AND NOT GVL.VS_S02_1 AND GVL.VS_S02_2 THEN
	
		IF GVL.volume_S02 > 0 AND GVL.volume_TQ2 < 25000 THEN
			GVL.volume_S02 := GVL.volume_S02 - GVL.V_S02_TQ;
			GVL.volume_TQ2 := GVL.volume_TQ2 + GVL.V_S02_TQ; // Diminuo o volume do tanque
			
		ELSIF GVL.volume_S02 > 0 AND GVL.volume_TQ2 >= 25000 THEN
			GVL.volume_S02 := GVL.volume_S02 - GVL.V_S02_TQ;
		END_IF
		
	ELSIF (GVL.D1_B_R2 OR GVL.D2_B_R2) AND NOT GVL.VA_S02 AND GVL.VS_S02_1 AND NOT GVL.VS_S02_2 THEN
	
		IF GVL.volume_S02 > 0 AND GVL.volume_TQ1 < 25000 THEN
			GVL.volume_S02 := GVL.volume_S02 - GVL.V_S02_TQ;
			GVL.volume_TQ1 := GVL.volume_TQ1 + GVL.V_S02_TQ; // Diminuo o volume do tanque
			
		ELSIF GVL.volume_S02 > 0 AND GVL.volume_TQ1 >= 25000 THEN
			GVL.volume_S02 := GVL.volume_S02 - GVL.V_S02_TQ;
		END_IF
	
	ELSIF (GVL.D1_B_R2 OR GVL.D2_B_R2) AND NOT GVL.VA_S02 AND GVL.VS_S02_1 AND GVL.VS_S02_2 THEN
		
			IF GVL.volume_S02 > 0 AND GVL.volume_TQ1 < 25000 AND GVL.volume_TQ2 < 25000 THEN
				GVL.volume_S02 := GVL.volume_S02 - GVL.V_S02_TQ;
				GVL.volume_TQ1 := GVL.volume_TQ1 + GVL.V_S02_TQ; // Diminuo o volume do tanque
				GVL.volume_TQ2 := GVL.volume_TQ2 + GVL.V_S02_TQ;
				
			ELSIF GVL.volume_S02 > 0 AND GVL.volume_TQ1 >= 25000 AND GVL.volume_TQ2 < 25000 THEN
				GVL.volume_S02 := GVL.volume_S02 - GVL.V_S02_TQ;
				GVL.volume_TQ2 := GVL.volume_TQ2 + GVL.V_S02_TQ;
				
			ELSIF GVL.volume_S02 > 0 AND GVL.volume_TQ1 < 25000 AND GVL.volume_TQ2 >= 25000 THEN
				GVL.volume_S02 := GVL.volume_S02 - GVL.V_S02_TQ;
				GVL.volume_TQ1 := GVL.volume_TQ1 + GVL.V_S02_TQ;
				
			ELSIF GVL.volume_S02 > 0 AND GVL.volume_TQ1 >= 25000 AND GVL.volume_TQ2 >= 25000 THEN
				GVL.volume_S02 := GVL.volume_S02 - GVL.V_S02_TQ;
				
			END_IF
		
	ELSIF (GVL.D1_B_R2 OR GVL.D2_B_R2) AND GVL.VA_S02 AND NOT GVL.VS_S02_1 AND NOT GVL.VS_S02_2 THEN
	
		IF GVL.volume_S02 < 50000 THEN
			GVL.volume_S02 := GVL.volume_S02 + GVL.V_R_Gasolina;
	
		ELSIF GVL.volume_S02 >= 50000 THEN
			GVL.Transbordo_S02 := TRUE;
		END_IF
		
	ELSIF (GVL.D1_B_R2 OR GVL.D2_B_R2) AND GVL.VA_S02 AND GVL.VS_S02_1 AND NOT GVL.VS_S02_2 THEN	
		
		IF GVL.volume_S02 < 50000 AND GVL.volume_TQ1 < 25000 THEN	
	
			GVL.volume_S02 := GVL.volume_S02 + GVL.V_R_Gasolina;
			GVL.volume_S02 := GVL.volume_S02 - GVL.V_S02_TQ;
			GVL.volume_TQ1 := GVL.volume_TQ1 + GVL.V_S02_TQ;
			
		ELSIF GVL.volume_S02 < 50000 AND GVL.volume_TQ1 >= 25000 THEN
			
			GVL.volume_S02 := GVL.volume_S02 + GVL.V_R_Gasolina;
			
			
		ELSIF GVL.volume_S02 >= 50000 AND GVL.volume_TQ1 < 25000 THEN
			
			GVL.Transbordo_S02 := TRUE;
			GVL.volume_S02 := GVL.volume_S02 - GVL.V_S02_TQ;
			GVL.volume_TQ1 := GVL.volume_TQ1 + GVL.V_S02_TQ;
			
		ELSIF GVL.volume_S01 >= 50000  AND GVL.volume_TQ1 >= 25000 THEN
			GVL.Transbordo_S02 := TRUE;

		END_IF
	ELSIF (GVL.D1_B_R2 OR GVL.D2_B_R2) AND GVL.VA_S02 AND NOT GVL.VS_S02_1 AND GVL.VS_S02_2 THEN	
		
		IF GVL.volume_S02 < 50000 AND GVL.volume_TQ2 < 25000 THEN	
	
			GVL.volume_S02 := GVL.volume_S02 + GVL.V_R_Gasolina;
			GVL.volume_S02 := GVL.volume_S02 - GVL.V_S02_TQ;
			GVL.volume_TQ2 := GVL.volume_TQ2 + GVL.V_S02_TQ;
			
		ELSIF GVL.volume_S02 < 50000 AND GVL.volume_TQ2 >= 25000 THEN
			
			GVL.volume_S02 := GVL.volume_S02 + GVL.V_R_Gasolina;
			
			
		ELSIF GVL.volume_S02 >= 50000 AND GVL.volume_TQ2 < 25000 THEN
			
			GVL.Transbordo_S02 := TRUE;
			GVL.volume_S02 := GVL.volume_S02 - GVL.V_S02_TQ;
			GVL.volume_TQ2 := GVL.volume_TQ2 + GVL.V_S02_TQ;
			
		ELSIF GVL.volume_S01 >= 50000  AND GVL.volume_TQ2 >= 25000 THEN
			GVL.Transbordo_S02 := TRUE;

		END_IF
	
	ELSIF (GVL.D1_B_R2 OR GVL.D2_B_R2) AND GVL.VA_S02 AND GVL.VS_S02_1 AND GVL.VS_S02_2 THEN	
		
		IF GVL.volume_S02 < 50000 AND GVL.volume_TQ2 < 25000 AND GVL.volume_TQ1 < 25000 THEN	
	
			GVL.volume_S02 := GVL.volume_S02 + GVL.V_R_Gasolina;
			GVL.volume_S02 := GVL.volume_S02 - GVL.V_S02_TQ;
			GVL.volume_S02 := GVL.volume_S02 - GVL.V_S02_TQ;
			GVL.volume_TQ1 := GVL.volume_TQ1 + GVL.V_S02_TQ;
			GVL.volume_TQ2 := GVL.volume_TQ2 + GVL.V_S02_TQ;
		
		ELSIF GVL.volume_S02 < 50000 AND GVL.volume_TQ2 < 25000 AND GVL.volume_TQ1 >= 25000 THEN	
			
			GVL.volume_S02 := GVL.volume_S02 + GVL.V_R_Gasolina;
			GVL.volume_S02 := GVL.volume_S02 - GVL.V_S02_TQ;
			GVL.volume_TQ2 := GVL.volume_TQ2 + GVL.V_S02_TQ;
		
		ELSIF GVL.volume_S02 < 50000 AND GVL.volume_TQ2 >= 25000 AND GVL.volume_TQ1 < 25000 THEN	
			
			GVL.volume_S02 := GVL.volume_S02 + GVL.V_R_Gasolina;
			GVL.volume_S02 := GVL.volume_S02 - GVL.V_S02_TQ;
			GVL.volume_TQ1 := GVL.volume_TQ1 + GVL.V_S02_TQ;	
			
		ELSIF GVL.volume_S02 < 50000 AND GVL.volume_TQ2 >= 25000 AND GVL.volume_TQ1 >= 25000 THEN	
			
			GVL.volume_S02 := GVL.volume_S02 + GVL.V_R_Gasolina;	
			
		ELSIF GVL.volume_S02 >= 50000 AND GVL.volume_TQ2 < 25000 AND GVL.volume_TQ1 < 25000 THEN
			
			GVL.Transbordo_S02 := TRUE;
			GVL.volume_S02 := GVL.volume_S02 - GVL.V_S02_TQ;
			GVL.volume_S02 := GVL.volume_S02 - GVL.V_S02_TQ;
			GVL.volume_TQ1 := GVL.volume_TQ1 + GVL.V_S02_TQ;
			GVL.volume_TQ2 := GVL.volume_TQ2 + GVL.V_S02_TQ;
			
		ELSIF GVL.volume_S02 >= 50000 AND GVL.volume_TQ2 < 25000 AND GVL.volume_TQ1 >= 25000 THEN
			
			GVL.Transbordo_S02 := TRUE;
			GVL.volume_S02 := GVL.volume_S02 - GVL.V_S02_TQ;
			GVL.volume_TQ2 := GVL.volume_TQ2 + GVL.V_S02_TQ;
			
			
		ELSIF GVL.volume_S02 >= 50000 AND GVL.volume_TQ2 >= 25000 AND GVL.volume_TQ1 < 25000 THEN
			
			GVL.Transbordo_S02 := TRUE;
			GVL.volume_S02 := GVL.volume_S02 - GVL.V_S02_TQ;
			GVL.volume_TQ1 := GVL.volume_TQ1 + GVL.V_S02_TQ;
			
			
		ELSIF GVL.volume_S02 >= 50000 AND GVL.volume_TQ2 >= 25000 AND GVL.volume_TQ1 >= 25000 THEN
			GVL.Transbordo_S02 := TRUE;

		END_IF	
		
	END_IF
END_IF

IF GVL.volume_S02 > 45000 AND GVL.VA_S02 AND (GVL.D1_B_R2 OR GVL.D1_B_R2) THEN
	
	GVL.LSH_S02 := TRUE;
	GVL.LSL_S02 := FALSE;
	
	GVL.ALARME_LSH_S02 := TRUE;
	GVL.ALARME_LSL_S02 := FALSE;
	
ELSIF GVL.volume_S02 < 5000 THEN
	
	GVL.LSH_S02 := FALSE;
	GVL.LSL_S02 := TRUE;
	
	GVL.ALARME_LSH_S02 := FALSE;
	GVL.ALARME_LSL_S02 := TRUE;
	
END_IF

IF (GVL.D1_B_R1 OR GVL.D2_B_R1) THEN
	GVL.B_R1 := TRUE;
ELSE
	GVL.B_R1 := FALSE;
END_IF

IF (GVL.D1_B_R2 OR GVL.D2_B_R2) THEN
	GVL.B_R2 := TRUE;
ELSE
	GVL.B_R2 := FALSE;
END_IF

END_PROGRAM

// Device/Application/Simulacao/Manual/Manual_Simulacao_Silo_01
PROGRAM Manual_Simulacao_Silo_01
VAR
END_VAR

IF NOT GVL.emergencia AND NOT GVL.switch THEN
	
	IF NOT GVL.D1_B_R1 AND NOT GVL.VS_S01 AND GVL.VC_TQ1 THEN	
	
		IF GVL.volume_TQ1 > 0 THEN
			
			GVL.volume_TQ1 := GVL.volume_TQ1 - GVL.TQ1_C; // Diminuo o volume do tanque
			
		END_IF
		
	ELSIF NOT GVL.D1_B_R1 AND GVL.VS_S01 AND NOT GVL.VC_TQ1 THEN
		
		IF GVL.volume_S01 > 0 AND GVL.volume_TQ1 < 25000 THEN
			GVL.volume_S01 := GVL.volume_S01 - GVL.V_S01_TQ1; //Diminuo o volume do silo
		
			GVL.volume_TQ1 := GVL.volume_TQ1 + GVL.V_S01_TQ1; // Aumento o volume do tanque
		END_IF
	
	ELSIF NOT GVL.D1_B_R1 AND GVL.VS_S01 AND GVL.VC_TQ1 THEN
		
		IF GVL.volume_S01 > 0 THEN
			GVL.volume_S01 := GVL.volume_S01 - GVL.V_S01_TQ1; //Diminuo o volume do silo
			GVL.volume_TQ1 := GVL.volume_TQ1 + GVL.V_S01_TQ1 - GVL.TQ1_C;;
		ELSIF GVL.volume_TQ1 > 0 THEN
			GVL.volume_TQ1 := GVL.volume_TQ1 - GVL.TQ1_C; // Mantenho o volume do tanque, 
		END_IF
		
	ELSIF GVL.D1_B_R1 AND NOT GVL.VA_S01 AND NOT GVL.VS_S01 AND GVL.VC_TQ1 THEN
		
		IF GVL.volume_TQ1 > 0 THEN
			
			GVL.volume_TQ1 := GVL.volume_TQ1 - GVL.TQ1_C; // Diminuo o volume do tanque
			
		END_IF
		
	ELSIF GVL.D1_B_R1 AND NOT GVL.VA_S01 AND GVL.VS_S01 AND NOT GVL.VC_TQ1 THEN
	
		IF GVL.volume_S01 > 0 AND GVL.volume_TQ1 < 25000 THEN
			
			GVL.volume_S01 := GVL.volume_S01 - GVL.V_S01_TQ1; //Diminuo o volume do silo
		
			GVL.volume_TQ1 := GVL.volume_TQ1 + GVL.V_S01_TQ1; // Aumento o volume do tanque
		END_IF
	
	ELSIF GVL.D1_B_R1 AND NOT GVL.VA_S01 AND GVL.VS_S01 AND GVL.VC_TQ1 THEN
	
		IF GVL.volume_S01 > 0 THEN
			GVL.volume_S01 := GVL.volume_S01 - GVL.V_S01_TQ1; //Diminuo o volume do silo
			GVL.volume_TQ1 := GVL.volume_TQ1 + GVL.V_S01_TQ1 - GVL.TQ1_C;;
		ELSIF GVL.volume_TQ1 > 0 THEN
			GVL.volume_TQ1 := GVL.volume_TQ1 - GVL.TQ1_C; // Mantenho o volume do tanque, 
		END_IF	
		
	ELSIF GVL.D1_B_R1 AND GVL.VA_S01 AND NOT GVL.VS_S01 AND NOT GVL.VC_TQ1 THEN	
		IF GVL.volume_S01 < 50000 THEN		
			GVL.volume_S01 := GVL.volume_S01 + GVL.V_S01_TQ1;
		ELSIF GVL.volume_S01 >= 50000 THEN
			GVL.Transbordo_S01 := TRUE;
		END_IF
		
	ELSIF GVL.D1_B_R1 AND GVL.VA_S01 AND NOT GVL.VS_S01 AND NOT GVL.VC_TQ1 THEN	
		IF GVL.volume_S01 < 50000 THEN		
			GVL.volume_S01 := GVL.volume_S01 + GVL.V_S01_TQ1;
		ELSIF GVL.volume_S01 >= 50000 THEN
			GVL.Transbordo_S01 := TRUE;
		END_IF
		
	ELSIF GVL.D1_B_R1 AND GVL.VA_S01 AND NOT GVL.VS_S01 AND GVL.VC_TQ1 THEN	
		
		IF GVL.volume_S01 < 50000 AND GVL.volume_TQ1 > 0 THEN	
	
			GVL.volume_S01 := GVL.volume_S01 + GVL.V_R_Etanol;
			GVL.volume_TQ1 := GVL.volume_TQ1 - GVL.TQ1_C;
			
		ELSIF GVL.volume_S01 < 50000 AND GVL.volume_TQ1 < 0 THEN
			
			GVL.volume_S01 := GVL.volume_S01 + GVL.V_R_Etanol;
			
		ELSIF GVL.volume_S01 >= 50000 AND GVL.volume_TQ1 > 0 THEN
			
			GVL.Transbordo_S01 := TRUE;
			GVL.volume_TQ1 := GVL.volume_TQ1 - GVL.TQ1_C;
			
		ELSIF GVL.volume_S01 >= 50000  AND GVL.volume_TQ1 < 0 THEN
			GVL.Transbordo_S01 := TRUE;
		END_IF
	
	ELSIF GVL.D1_B_R1 AND GVL.VA_S01 AND GVL.VS_S01 AND NOT GVL.VC_TQ1 THEN	
		
		IF GVL.volume_S01 < 50000 AND GVL.volume_TQ1 < 25000  THEN	
	
			GVL.volume_S01 := GVL.volume_S01 + GVL.V_R_Etanol;
			GVL.volume_S01 := GVL.volume_S01 - GVL.V_S01_TQ1;
			GVL.volume_TQ1 := GVL.volume_TQ1 + GVL.V_S01_TQ1;
			
		ELSIF GVL.volume_S01 >= 50000 AND GVL.volume_TQ1 < 25000  THEN	
			
			GVL.Transbordo_S01 := TRUE;
			GVL.volume_TQ1 := GVL.volume_TQ1 + GVL.V_S01_TQ1;
			
		ELSIF GVL.volume_S01 < 50000 AND GVL.volume_TQ1 > 25000 THEN
			
			GVL.volume_S01 := GVL.volume_S01 + GVL.V_R_Etanol;
			
		ELSIF GVL.volume_S01 >= 50000 AND GVL.volume_TQ1 >25000 THEN
			
			GVL.Transbordo_S01 := TRUE;
			
		END_IF
	
	ELSIF GVL.D1_B_R1 AND GVL.VA_S01 AND GVL.VS_S01 AND GVL.VC_TQ1 THEN		
		
		IF GVL.volume_S01 < 50000 AND GVL.volume_TQ1 < 25000  THEN	
	
			GVL.volume_S01 := GVL.volume_S01 + GVL.V_R_Etanol;
			GVL.volume_S01 := GVL.volume_S01 - GVL.V_S01_TQ1;
			GVL.volume_TQ1 := GVL.volume_TQ1 + GVL.V_S01_TQ1;
			GVL.volume_TQ1 := GVL.volume_TQ1 - GVL.TQ1_C;
			
		ELSIF GVL.volume_S01 >= 50000 AND GVL.volume_TQ1 < 25000  THEN	
			
			GVL.Transbordo_S01 := TRUE;
			GVL.volume_TQ1 := GVL.volume_TQ1 + GVL.V_S01_TQ1;
			GVL.volume_TQ1 := GVL.volume_TQ1 - GVL.TQ1_C;
			
		ELSIF GVL.volume_S01 < 50000 AND GVL.volume_TQ1 > 25000 THEN
			
			GVL.volume_S01 := GVL.volume_S01 + GVL.V_R_Etanol;
			
		ELSIF GVL.volume_S01 >= 50000 AND GVL.volume_TQ1 >25000 THEN
			
			GVL.Transbordo_S01 := TRUE;
			
		END_IF
		
	END_IF
END_IF

IF GVL.volume_S01 > 45000 AND GVL.VA_S01 AND (GVL.D1_B_R1 OR GVL.D1_B_R1) THEN
	
	GVL.LSH_S01 := TRUE;
	GVL.LSL_S01 := FALSE;
	
	GVL.ALARME_LSH_S01 := TRUE;
	GVL.ALARME_LSL_S01 := FALSE;
	
ELSIF GVL.volume_S01 < 5000 THEN
	
	GVL.LSH_S01 := FALSE;
	GVL.LSL_S01 := TRUE;
	
	GVL.ALARME_LSH_S01 := FALSE;
	GVL.ALARME_LSL_S01 := TRUE;
	
END_IF

IF (GVL.D1_B_R1 OR GVL.D2_B_R1) THEN
	GVL.B_R1 := TRUE;
ELSE
	GVL.B_R1 := FALSE;
END_IF

IF (GVL.D1_B_R2 OR GVL.D2_B_R2) THEN
	GVL.B_R2 := TRUE;
ELSE
	GVL.B_R2 := FALSE;
END_IF

END_PROGRAM

// Device/Application/Simulacao/Automatico/Valores_Doca2_Simulacao
PROGRAM Valores_Doca2_Simulacao
VAR
	Volume_gasolina_comum : REAL := 25000 * 0.75;
	Volume_etanol_comum : REAL := 25000 * 0.25;
	Volume_gasolina_premium : REAL := 25000 * 0.73;
	Volume_etanol_premium : REAL := 25000 * 0.27;
END_VAR

IF GVL.volume_C2 >= 25000 THEN // AND GVL.volume_gasolina_C2 = 0 THEN
	Doca2_automatico.etanol_cheio := TRUE;
	GVL.caminhao2_cheio := TRUE;
	
	GVL.volume_etanol_C2 := 0;
	GVL.volume_gasolina_C2 := 0;
	
ELSIF GVL.volume_S03 <= 5000 THEN
	GVL.LSL_S03 := TRUE;
	GVL.LSH_S03 := FALSE;

ELSIF  GVL.volume_S02 <= 5000 THEN
	GVL.LSL_S02 := TRUE;
	GVL.LSH_S02 := FALSE;

ELSIF GVL.volume_S02 >= 45000 AND GVL.B_R2 THEN
	GVL.LSH_S02 := TRUE;
	GVL.LSL_S02 := FALSE;
	
ELSIF GVL.volume_S03 >= 45000 AND GVL.B_R1 THEN
	GVL.LSH_S03 := TRUE;
	GVL.LSL_S03 := FALSE;

ELSIF GVL.volume_etanol_C2 >= Volume_etanol_premium AND NOT (GVL.volume_gasolina_C2 >= Volume_gasolina_premium) AND GVL.PREMIUM THEN // PODE GERAR UM FUTURO PROBLEMA
	Doca2_automatico.etanol_cheio := TRUE;	
	
ELSIF GVL.volume_gasolina_C2 >= Volume_gasolina_premium AND NOT GVL.M2 AND GVL.PREMIUM THEN // PODE GERAR UM PROBLEMA NO FUTURO	
	Doca2_automatico.gasolina_cheio := TRUE;
	
ELSIF GVL.volume_etanol_C2 >= Volume_etanol_comum AND NOT (GVL.volume_gasolina_C2 >= Volume_gasolina_comum) AND NOT GVL.PREMIUM THEN // PODE GERAR UM FUTURO PROBLEMA
	Doca2_automatico.etanol_cheio := TRUE;
	
ELSIF GVL.volume_gasolina_C2 >= Volume_gasolina_comum AND NOT GVL.M2 AND NOT GVL.PREMIUM THEN // PODE GERAR UM PROBLEMA NO FUTURO
	Doca2_automatico.gasolina_cheio := TRUE;
	
ELSIF GVL.M2 THEN
	GVL.volume_etanol_C2 := 0;
	GVL.volume_gasolina_C2 := 0;
	
ELSE
	GVL.LSL_S03 := FALSE;
	GVL.caminhao2_cheio := FALSE;
	Doca2_automatico.etanol_cheio := FALSE;
	Doca2_automatico.gasolina_cheio := FALSE;
	GVL.LSH_S03 := FALSE;
END_IF

END_PROGRAM

// Device/Application/Simulacao/Automatico/Valores_Doca1_Simulacao
PROGRAM Valores_Doca1_Simulacao
VAR
	Volume_gasolina_comum : REAL := 25000 * 0.75;
	Volume_etanol_comum : REAL := 25000 * 0.25;
	Volume_gasolina_premium : REAL := 25000 * 0.73;
	Volume_etanol_premium : REAL := 25000 * 0.27;
END_VAR

IF GVL.volume_C1 >= 25000 THEN//AND GVL.volume_gasolina_C1 = 0 THEN
	Doca1_automatico.etanol_cheio := TRUE;
	GVL.caminhao1_cheio := TRUE;
	
	GVL.volume_etanol_C1 := 0;
	GVL.volume_gasolina_C1 := 0;
	
ELSIF GVL.volume_S01 <= 5000 THEN
	GVL.LSL_S01 := TRUE;
	GVL.LSH_S01 := FALSE;
	
ELSIF  GVL.volume_S02 <= 5000 THEN
	GVL.LSL_S02 := TRUE;
	GVL.LSH_S02 := FALSE;

ELSIF GVL.volume_S02 >= 45000 AND GVL.B_R2 THEN
	GVL.LSH_S02 := TRUE;
	GVL.LSL_S02 := FALSE;
	
ELSIF GVL.volume_S01 >= 45000 AND GVL.B_R1 THEN
	GVL.LSH_S01 := TRUE;
	GVL.LSL_S01 := FALSE;

ELSIF GVL.volume_etanol_C1 >= Volume_etanol_premium AND NOT (GVL.volume_gasolina_C1 >= Volume_gasolina_premium) AND GVL.PREMIUM THEN // PODE GERAR UM FUTURO PROBLEMA
	Doca1_automatico.etanol_cheio := TRUE;
	
ELSIF GVL.volume_gasolina_C1 >= Volume_gasolina_premium AND NOT GVL.M1 AND GVL.PREMIUM THEN // PODE GERAR UM PROBLEMA NO FUTURO
	Doca1_automatico.gasolina_cheio := TRUE;	
	
ELSIF GVL.volume_etanol_C1 >= Volume_etanol_comum AND NOT (GVL.volume_gasolina_C1 >= Volume_gasolina_comum) AND NOT GVL.PREMIUM THEN // PODE GERAR UM FUTURO PROBLEMA
	Doca1_automatico.etanol_cheio := TRUE;
	
ELSIF GVL.volume_gasolina_C1 >= Volume_gasolina_comum AND NOT GVL.M1 AND NOT GVL.PREMIUM THEN // PODE GERAR UM PROBLEMA NO FUTURO
	Doca1_automatico.gasolina_cheio := TRUE;
	
ELSIF GVL.M1 THEN
	GVL.volume_etanol_C1 := 0;
	GVL.volume_gasolina_C1 := 0;
	
ELSE
	GVL.LSL_S01 := FALSE;
	GVL.caminhao1_cheio := FALSE;
	Doca1_automatico.gasolina_cheio := FALSE;
	Doca1_automatico.etanol_cheio := FALSE;
	GVL.LSH_S01 := FALSE;
END_IF

IF (GVL.D1_B_R1 OR GVL.D2_B_R1) THEN
	GVL.B_R1 := TRUE;
ELSE
	GVL.B_R1 := FALSE;
END_IF

IF (GVL.D1_B_R2 OR GVL.D2_B_R2) THEN
	GVL.B_R2 := TRUE;
ELSE
	GVL.B_R2 := FALSE;
END_IF

END_PROGRAM

// Valores_Simulacao_Manual
PROGRAM Valores_Simulacao_Manual
VAR
END_VAR

IF NOT GVL.emergencia AND NOT GVL.switch THEN

	IF GVL.Y_C_D1 AND GVL.Y_M_D1 AND GVL.VC_TQ1 AND (GVL.volume_TQ1 > 0  OR GVL.VS_S01 OR GVL.VS_S02_1) AND NOT GVL.Y_C_D2 AND NOT GVL.Y_M_D2 AND NOT GVL.VC_TQ2 THEN
		
		IF GVL.volume_C1 < 25000 THEN
			GVL.volume_C1 := GVL.volume_C1 + GVL.TQ1_C;		
		END_IF
		
	ELSIF NOT GVL.Y_C_D1 AND NOT GVL.Y_M_D1 AND NOT GVL.VC_TQ1 AND GVL.Y_C_D2 AND GVL.Y_M_D2 AND GVL.VC_TQ2 AND (GVL.volume_TQ2 > 0  OR GVL.VS_S03 OR GVL.VS_S02_2) THEN 
		
		IF GVL.volume_C2 < 25000 THEN
			GVL.volume_C2 := GVL.volume_C2 + GVL.TQ2_C;
		END_IF
		
	ELSIF GVL.Y_C_D1 AND GVL.Y_M_D1 AND GVL.VC_TQ1 AND GVL.Y_C_D2 AND GVL.Y_M_D2 AND GVL.VC_TQ2 AND (GVL.volume_TQ1 > 0  OR GVL.VS_S01 OR GVL.VS_S02_1) AND (GVL.volume_TQ2 > 0  OR GVL.VS_S03 OR GVL.VS_S02_2) THEN
		
		IF GVL.volume_C2 < 25000 AND GVL.volume_C1 < 25000 THEN
			
			GVL.volume_C1 := GVL.volume_C1 + GVL.TQ1_C;
			GVL.volume_C2 := GVL.volume_C2 + GVL.TQ2_C;
			
		ELSIF GVL.volume_C2 < 25000 AND GVL.volume_C1 >= 25000 THEN
			
			GVL.volume_C2 := GVL.volume_C2 + GVL.TQ2_C;
			
		ELSIF GVL.volume_C1 < 25000 AND GVL.volume_C2 >= 25000 THEN
			
			GVL.volume_C1 := GVL.volume_C1 + GVL.TQ1_C;	
			
		END_IF
	ELSIF NOT GVL.Y_C_D1 AND NOT GVL.Y_M_D1  AND NOT GVL.Y_C_D2 AND NOT GVL.Y_M_D2 THEN
		
		GVL.volume_C1 := 0;	
		GVL.volume_C2 := 0;
		
	ELSIF NOT GVL.Y_C_D1 AND NOT GVL.Y_M_D1 AND GVL.Y_C_D2 AND GVL.Y_M_D2 THEN 
		
		GVL.volume_C1 := 0;	
	
	ELSIF GVL.Y_C_D1 AND GVL.Y_M_D1 AND NOT GVL.Y_C_D2 AND NOT GVL.Y_M_D2 THEN 	
		
		GVL.volume_C2 := 0;
	
	END_IF
END_IF

END_PROGRAM

// Device/Application/Alarmes
PROGRAM Alarmes
VAR
END_VAR

END_PROGRAM
